# EPICS substitutions: src/makeBaseApp/top/pcdsMotorApp/Db/motors.substitutions
# P, M, and N combine to make the instance's name.
# N contains the specific motor.
# DTYP is the motor driver name for our motors.
# C is controller; this links to the ASYN port
#   ASYN gives digi port a name
#   MDrivePlusConfig maps digi name to controller #.
# ACCL is the time to accelerate from the base speed to full speed.
# DIR is the direction of rotation, "Pos" or "Neg"

# SREV (not shown) is the number of steps per revolution is 200 by
#    default
#

#
# For SREV:
#    2048 = internal encoder (EQ)
#     250 = external encoder, NUMERIK-JENA
#     200 = external encoder, Renishaw
#   51200 = no encoder

# NOTE: Soft limits (DHLM & DLLM) may be better off using HLM & LLM and relying on autosave to keep those than loading them into the database everytime.
# If the motor is reversed in DIR, then the DHLM and HLM are reveresed which makes it difficult to accurately set the soft limits.
# (Dial) DHLM 140, DLLM 2 is equivalent to (User) HLM -2, LLM -140

file basic_motor_jt.template
{
pattern
   {P,                  M,  DTYP,         C,  S, DESC,                     EGU, DIR, SREV,  UREV,    SP,    SBAS,  SMAX,  ACCL,  RDBD, DLY, PREC, DHLM,  DLLM}
   {$(LOC):$(SYS):MMS:, 01, "MDrivePlus", 0,  0, "Manipulator 1 X",        mm,  Neg, 51200, 2.116,   1,     0.098, 1,     0.1,   0.01, 0,   4,    5.0,   -5.0}
#   {$(LOC):$(SYS):MMS:, 02, "MDrivePlus", 1,  0, "Manipulator 1 Y",        mm,  Pos, 51200, 2.116,   1,     0.098, 1,     0.1,   0.01, 0,   4,    5.0,   -5.0}
}

file motor-status.template
{
pattern
   { MOT,                    DESC,				FW_MEANS,	REV_MEANS	}
   { "$(LOC):$(SYS):MMS:01", "Manipulator 1 X",	"X+",		"X-"		}
#  { "$(LOC):$(SYS):MMS:02", "Manipulator 1 Y",	"Y+",		"Y-"		}
}
